(* PLC project Unnamed, Unknown Unnamed 1 *)
(* stored: creationDateTime 2023-09-01T17:29:03, modificationDateTime 2023-09-06T13:29:42 *)

PROGRAM car_wash
  VAR
    conveyor_motor AT %QX0.0 : BOOL := False;
    washer_1 AT %QX0.1 : BOOL := False;
    washer_2 AT %QX0.2 : BOOL := False;
    brush_1 AT %QX0.3 : BOOL := False;
    brush_2 AT %QX0.4 : BOOL := False;
    rinse_1 AT %QX0.5 : BOOL := False;
    rinse_2 AT %QX0.6 : BOOL := False;
    dryer_1 AT %QX0.7 : BOOL := False;
    dryer_2 AT %QX1.0 : BOOL := False;
    in_use_light AT %QX1.1 : BOOL := False;
    wash_complete_light AT %QX1.2 : BOOL := False;
    master_start AT %QX1.3 : BOOL;
    master_stop AT %QX1.4 : BOOL;
    entry_sensor AT %QX1.5 : BOOL := False;
    was_sensor AT %QX1.6 : BOOL := False;
    brush_sensor AT %QX1.7 : BOOL := False;
    rinse_sensor AT %QX2.0 : BOOL := False;
    dry_sensor AT %QX2.1 : BOOL := False;
    exit_sensor AT %QX2.2 : BOOL := False;
    master_coil AT %QX2.3 : BOOL;
    conveyor_start_delay AT %QX2.4 : BOOL;
    washing_time AT %QX2.5 : BOOL;
    brushing_time AT %QX2.6 : BOOL;
    rinsing_time AT %QX2.7 : BOOL;
    drying_time AT %QX3.0 : BOOL;
  END_VAR
  VAR
    TON0 : TON;
    conveyor_delay_pt : TIME := T#5s;
    TON1 : TON;
    wash_time_pt : TIME := T#5s;
    TON2 : TON;
    brush_time_pt : TIME := T#5s;
    TON3 : TON;
    rinse_time_pt : TIME := T#5s;
    TON4 : TON;
    dry_time_pt : TIME := T#5s;
    exit_delay : TIME := T#3s;
  END_VAR

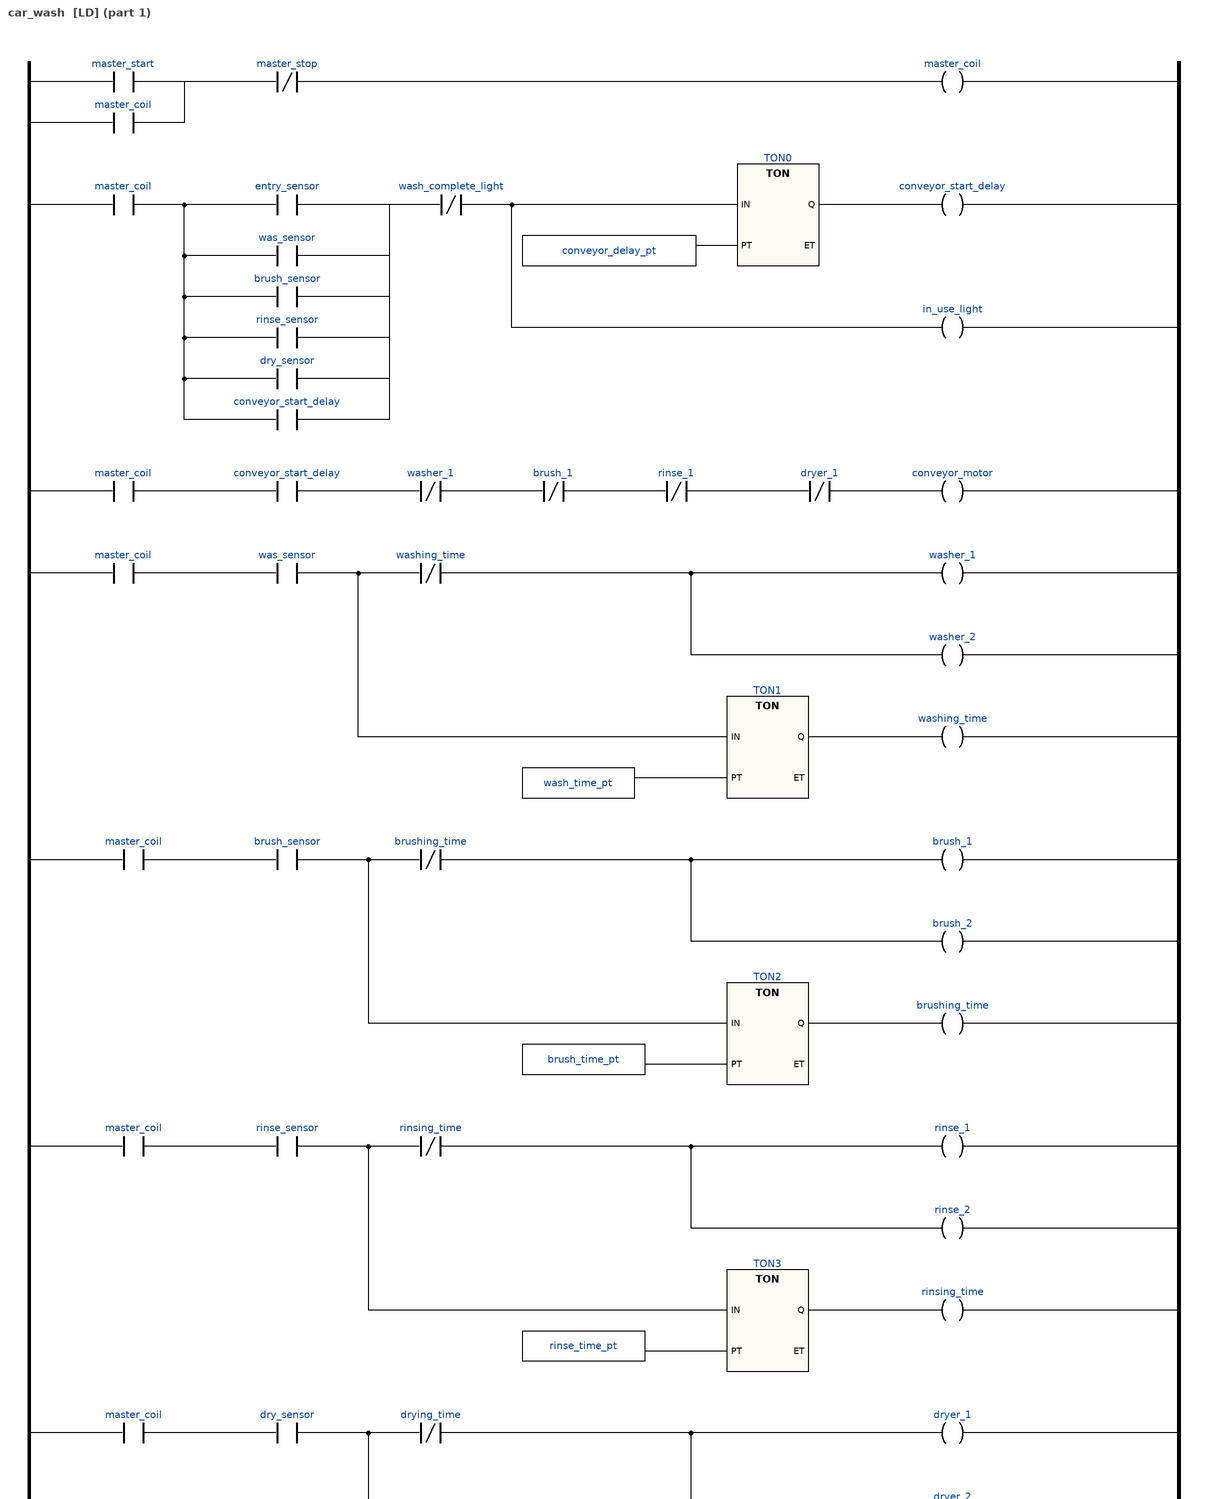
(* LD diagram, written out as Structured Text *)
master_coil := (master_start OR master_coil) AND NOT master_stop;
TON0(IN := master_coil AND (entry_sensor OR was_sensor OR brush_sensor OR rinse_sensor OR dry_sensor OR conveyor_start_delay) AND NOT wash_complete_light, PT := conveyor_delay_pt);
conveyor_start_delay := TON0.Q;
in_use_light := master_coil AND (entry_sensor OR was_sensor OR brush_sensor OR rinse_sensor OR dry_sensor OR conveyor_start_delay) AND NOT wash_complete_light;
conveyor_motor := master_coil AND conveyor_start_delay AND NOT washer_1 AND NOT brush_1 AND NOT rinse_1 AND NOT dryer_1;
washer_1 := master_coil AND was_sensor AND NOT washing_time;
washer_2 := master_coil AND was_sensor AND NOT washing_time;
TON1(IN := master_coil AND was_sensor, PT := wash_time_pt);
washing_time := TON1.Q;
brush_1 := master_coil AND brush_sensor AND NOT brushing_time;
brush_2 := master_coil AND brush_sensor AND NOT brushing_time;
TON2(IN := master_coil AND brush_sensor, PT := brush_time_pt);
brushing_time := TON2.Q;
rinse_1 := master_coil AND rinse_sensor AND NOT rinsing_time;
rinse_2 := master_coil AND rinse_sensor AND NOT rinsing_time;
TON3(IN := master_coil AND rinse_sensor, PT := rinse_time_pt);
rinsing_time := TON3.Q;
dryer_1 := master_coil AND dry_sensor AND NOT drying_time;
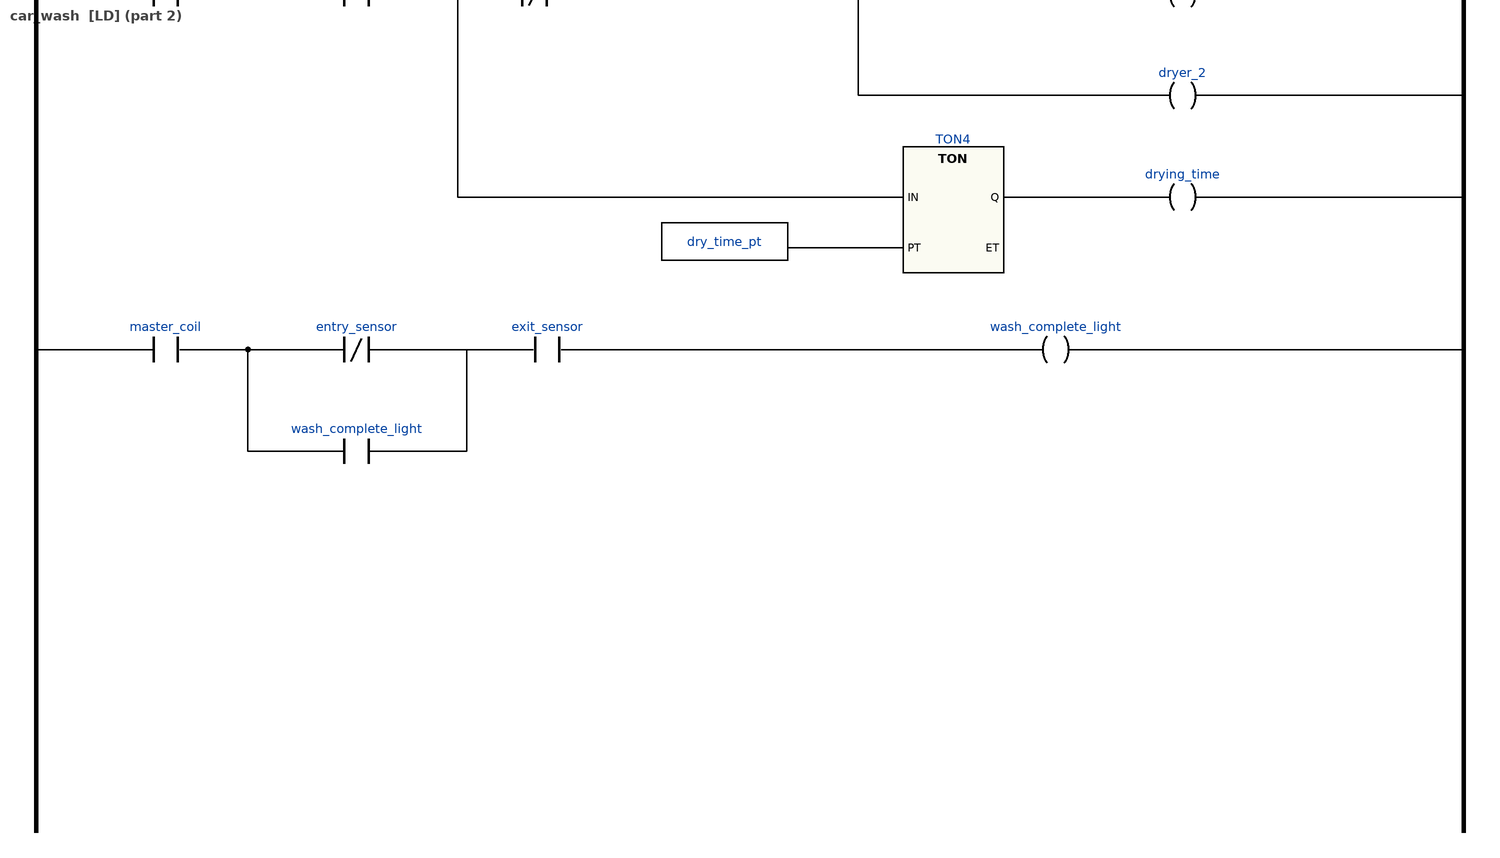
dryer_2 := master_coil AND dry_sensor AND NOT drying_time;
TON4(IN := master_coil AND dry_sensor, PT := dry_time_pt);
drying_time := TON4.Q;
wash_complete_light := master_coil AND (NOT entry_sensor OR wash_complete_light) AND exit_sensor;
END_PROGRAM

CONFIGURATION Config0
  RESOURCE Res0 ON PLC
    TASK task0(INTERVAL := T#20ms, PRIORITY := 0);
    PROGRAM instance0 WITH task0 : car_wash;
  END_RESOURCE
END_CONFIGURATION
